// TIA Portal V19 export
DATA_BLOCK "A0303_Spintore"   // DB95
// stored: InstanceOfName A0303_Spintore_FB, InstanceOfType FB
"A0303_Spintore_FB"
   // VAR_INPUT
   //    AreaInterface : "AreaInterface";
   //    ZSI : "udt_ZoneSafetyInterface";
   //    DSI : "udt_DeviceSafetyInterface";
   //    DataIn : Struct
   //       OP_Rest_PB : Bool;
   //       OP_Work_PB : Bool;
   //       LsPosition1 : Bool;
   //       LsMaxPosition : Bool;
   //    END_STRUCT;
   //    CIn : Struct
   //       Manager : Struct
   //          EnableStopDoorOpeningReq : Bool;
   //          EnableStopInPhase : Bool;
   //          EnableStopProgrammed : Bool;
   //          Control_ON : Bool;
   //          CanMoveFreely : Bool;
   //          Rest : Bool;
   //          Work : Bool;
   //       END_STRUCT;
   //       Manip : Struct
   //          OutOfWorkspace : Bool;
   //       END_STRUCT;
   //    END_STRUCT;
   //    Config : Struct
   //       Testa : Struct
   //          Vrt : "ValveMachine_Config";
   //          Orz : "ValveMachine_Config";
   //       END_STRUCT;
   //       Coda : Struct
   //          Vrt : "ValveMachine_Config";
   //          Orz : "ValveMachine_Config";
   //       END_STRUCT;
   //       DelayMissingCondition { ExternalAccessible := 'False'; ExternalVisible := 'False'; ExternalWritable := 'False'} : Time;
   //    END_STRUCT;
   // END_VAR
   // VAR_OUTPUT
   //    MachineInterface : "MachineInterface";
   //    COut : Struct
   //       Vrt : "ValveMachine_COut";
   //       Orz : "ValveMachine_COut";
   //    END_STRUCT;
   // END_VAR
   // VAR
   //    Alarm : Struct
   //       Testa : Struct
   //          Vrt : "ValveAlr";
   //          Orz : "ValveAlr";
   //       END_STRUCT;
   //       Coda : Struct
   //          Vrt : "ValveAlr";
   //          Orz : "ValveAlr";
   //       END_STRUCT;
   //       PassaggioPezzoNonOK : Bool;
   //    END_STRUCT;
   //    Warning : Struct
   //       Testa : Struct
   //          Vrt : "ValveMachine_Wng";
   //          Orz : "ValveMachine_Wng";
   //       END_STRUCT;
   //       Coda : Struct
   //          Vrt : "ValveMachine_Wng";
   //          Orz : "ValveMachine_Wng";
   //       END_STRUCT;
   //       OP_REST_MissingCnd : Bool;
   //       OP_WORK_MissingCnd : Bool;
   //    END_STRUCT;
   //    HMI : Struct
   //       Selection : Struct
   //          Vrt : Int;
   //          Orz : Int;
   //       END_STRUCT;
   //    END_STRUCT;
   //    Ctrl : Struct
   //       OP_Rest_Man : Bool;
   //       OP_Work_Man : Bool;
   //       OP_Rest_Aut : Bool;
   //       OP_Work_Aut : Bool;
   //       OP_Rest : Bool;
   //       OP_Work : Bool;
   //    END_STRUCT;
   //    Sts : Struct
   //       OP_Ax_CanMoveFreely : Bool;
   //       OP_Rest_Cnd : Bool;
   //       OP_Work_Cnd : Bool;
   //    END_STRUCT;
   //    Vrt_Testa : "ValveMachine_FB";
   //    Vrt_Coda : "ValveMachine_FB";
   //    Orz_Testa : "ValveMachine_FB";
   //    Orz_Coda : "ValveMachine_FB";
   //    AUX : Struct
   //       OP_Rest_PB { ExternalAccessible := 'False'; ExternalVisible := 'False'; ExternalWritable := 'False'} : Bool;
   //       OP_Work_PB { ExternalAccessible := 'False'; ExternalVisible := 'False'; ExternalWritable := 'False'} : Bool;
   //       LsPosition1_PE { ExternalAccessible := 'False'; ExternalVisible := 'False'; ExternalWritable := 'False'} : Bool;
   //       LsPosition1_NE { ExternalAccessible := 'False'; ExternalVisible := 'False'; ExternalWritable := 'False'} : Bool;
   //    END_STRUCT;
   //    TON_OP_REST_MissingCnd : IEC_TIMER;
   //    TON_OP_WORK_MissingCnd : IEC_TIMER;
   //    TON_CheckPos1Ok { S7_SetPoint := 'True'} : IEC_TIMER;
   // END_VAR
BEGIN
END_DATA_BLOCK
